// LS Electric XG5000 project: 66_1_A
// PLC NewPLC
// module base 0 slot 0: 입출력 모듈:XBC-DR20S (DC 24V 입력 12점, 릴레이 출력 8점)

PROGRAM NewProgram (task: 스캔 프로그램)

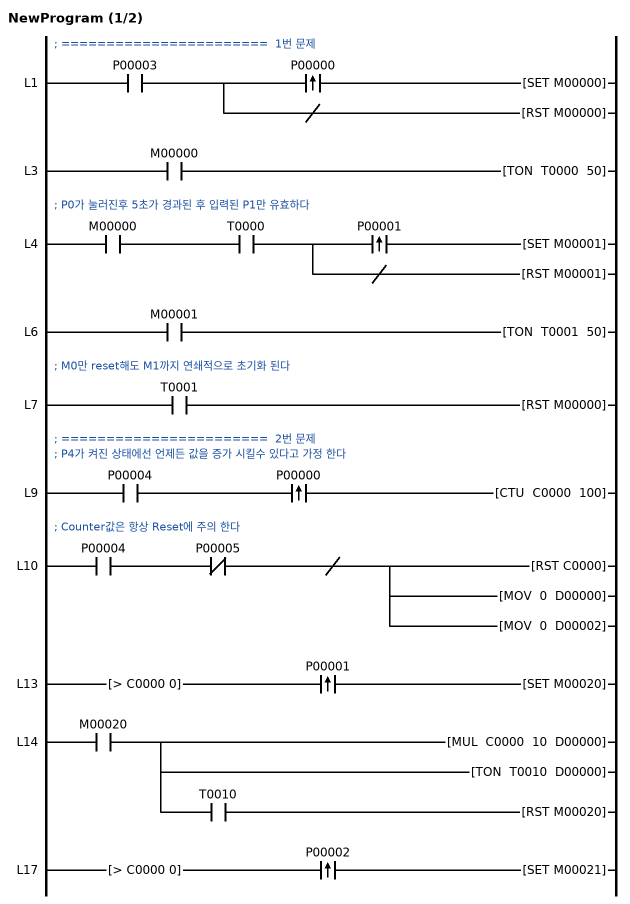
// =======================  1번 문제
; L1
LOAD      P00003
MPUSH
ANDP      P00000
SET       M00000
MPOP
NOT
RST       M00000
; L3
LOAD      M00000
TON       T0000 50
; L4
LOAD      M00000
AND       T0000
MPUSH
ANDP      P00001
SET       M00001
MPOP
NOT
RST       M00001
// output comment: P0가 눌러진후 5초가 경과된 후 입력된 P1만 유효하다
; L6
LOAD      M00001
TON       T0001 50
; L7
LOAD      T0001
RST       M00000
// output comment: M0만 reset해도 M1까지 연쇄적으로 초기화 된다
// =======================  2번 문제
; L9
LOAD      P00004
ANDP      P00000
CTU       C0000 100
// output comment: P4가 켜진 상태에선 언제든 값을 증가 시킬수 있다고 가정 한다
; L10
LOAD      P00004
AND NOT   P00005
NOT
RST       C0000
MOV       0 D00000
MOV       0 D00002
// output comment: Counter값은 항상 Reset에 주의 한다
; L13
LOAD>     C0000 0
ANDP      P00001
SET       M00020
; L14
LOAD      M00020
MUL       C0000 10 D00000
TON       T0010 D00000
AND       T0010
RST       M00020
; L17
LOAD>     C0000 0
ANDP      P00002
SET       M00021

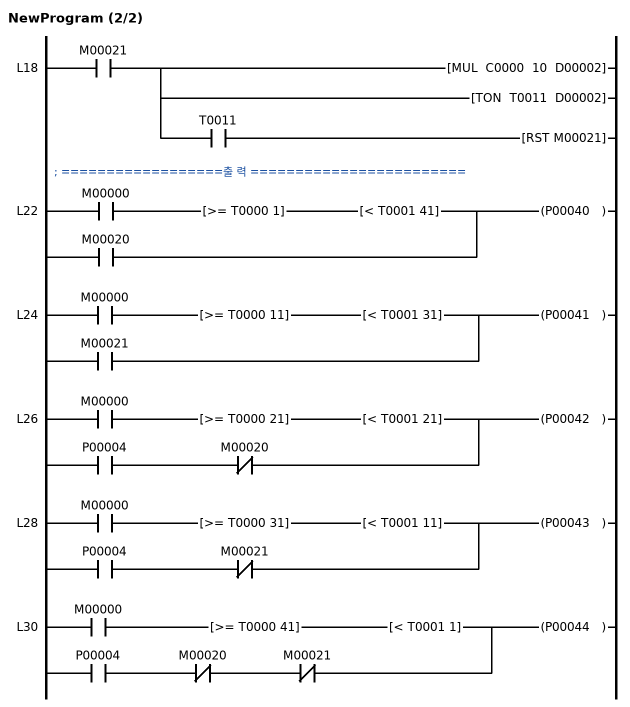
; L18
LOAD      M00021
MUL       C0000 10 D00002
TON       T0011 D00002
AND       T0011
RST       M00021
// ==================출 력 ========================
; L22
LOAD      M00000
AND>=     T0000 1
AND<      T0001 41
OR        M00020
OUT       P00040
; L24
LOAD      M00000
AND>=     T0000 11
AND<      T0001 31
OR        M00021
OUT       P00041
; L26
LOAD      M00000
AND>=     T0000 21
AND<      T0001 21
LOAD      P00004
AND NOT   M00020
OR LOAD
OUT       P00042
; L28
LOAD      M00000
AND>=     T0000 31
AND<      T0001 11
LOAD      P00004
AND NOT   M00021
OR LOAD
OUT       P00043
; L30
LOAD      M00000
AND>=     T0000 41
AND<      T0001 1
LOAD      P00004
AND NOT   M00020
AND NOT   M00021
OR LOAD
OUT       P00044